// TIA Portal V19 export
DATA_BLOCK "A0303_Sostegno_PERS"   // DB118
// stored: MemoryReserve 100
   VAR RETAIN
      Par : Struct
         Testa : Struct
            Ax : "Positioning_DOL_Machine_Par";
            Ax_Pers : "Positioning_DOL_Machine_Pers_Data";
            Enc : "PosFbk_RTN";
         END_STRUCT;
         Coda : Struct
            Ax : "Positioning_DOL_Machine_Par";
            Ax_Pers : "Positioning_DOL_Machine_Pers_Data";
            Enc : "PosFbk_RTN";
         END_STRUCT;
      END_STRUCT;
      Par_Mach : Struct
         RestPosition : LReal := 692.0;
         ToleranceWindow : LReal := 0.5;
         PosTimeout { ExternalVisible := 'False'} : Time := T#500MS;
      END_STRUCT;
   END_VAR
BEGIN
   Par.Testa.Ax.PosTolerance := 0.5;
   Par.Testa.Ax.Minus_Limit := 441.0;
   Par.Testa.Ax.Plus_Limit := 693.0;
   Par.Testa.Ax.PreCutOff := 0.2;
   Par.Testa.Ax.PreEndLowSpeed := 1.0;
   Par.Testa.Ax.PreEndMedSpeed := 10.0;
   Par.Testa.Ax.LowSpeed := 2.0;
   Par.Testa.Ax.MedSpeed := 15.0;
   Par.Testa.Ax.HighSpeed := 100.0;
   Par.Testa.Ax.Man_Speed := 100.0;
   Par.Testa.Ax_Pers.AxisHomed := TRUE;
   Par.Testa.Enc.Preset.Pulses := -958_761_696;
   Par.Testa.Enc.Preset.Units := 693.0;
   Par.Testa.Enc.Config.Resolution := 0.8;
   Par.Coda.Ax.PosTolerance := 0.5;
   Par.Coda.Ax.Minus_Limit := 441.0;
   Par.Coda.Ax.Plus_Limit := 693.0;
   Par.Coda.Ax.PreCutOff := 0.2;
   Par.Coda.Ax.PreEndLowSpeed := 1.0;
   Par.Coda.Ax.PreEndMedSpeed := 10.0;
   Par.Coda.Ax.LowSpeed := 2.0;
   Par.Coda.Ax.MedSpeed := 15.0;
   Par.Coda.Ax.HighSpeed := 100.0;
   Par.Coda.Ax.Man_Speed := 100.0;
   Par.Coda.Ax_Pers.AxisHomed := TRUE;
   Par.Coda.Enc.Preset.Pulses := -474_494_064;
   Par.Coda.Enc.Preset.Units := 693.0;
   Par.Coda.Enc.Config.Resolution := -0.8;
END_DATA_BLOCK
